// TwinCAT 3 PLC project PlcIotHttpSamplesTelegram
// ProgramVersion: 3.1.4026.25
// libraries:
//   Tc2_Standard, * (Beckhoff Automation GmbH)
//   Tc2_System, * (Beckhoff Automation GmbH)
//   Tc2_Utilities, * (Beckhoff Automation GmbH)
//   Tc3_IotBase, * (Beckhoff Automation GmbH)
//   Tc3_JsonXml, * (Beckhoff Automation GmbH)
//   Tc3_Module, * (Beckhoff Automation GmbH)
// project tree:
//   / PlcTask.TcTTO
//   POUs/ MAIN.TcPOU
//   POUs/Telegram/ FB_TestHTTP_Get_Telegram.TcPOU
// real-time tasks:
//   TASK PlcTask: cycle T#10ms, priority 25, ADS port 350

CONFIGURATION PlcIotHttpSamplesTelegram
    RESOURCE PLC ON TwinCAT3
        TASK PlcTask(INTERVAL := T#10ms, PRIORITY := 25);
        PROGRAM MAIN WITH PlcTask : MAIN;
    END_RESOURCE
END_CONFIGURATION

// ---- POUs/MAIN.TcPOU
PROGRAM MAIN
VAR
	// trigger command execution for Telegram samples
	bGetTelegram					: BOOL;

	fbHttpClientTelegram			: FB_IotHttpClient :=(sHostName := 'api.telegram.org',
									bKeepAlive := FALSE, tConnectionTimeout := T#10S);

	fbHttpGetTelegram				: FB_TestHTTP_Get_Telegram;
	sMessage						: STRING(500) := 'Hello from TwinCAT';
END_VAR

// init client parameters at startup
IF NOT fbHttpClientTelegram.bConfigured THEN
	fbHttpClientTelegram.nHostPort := 443;
	fbHttpClientTelegram.stTLS.bNoServerCertCheck := TRUE;
END_IF

IF fbHttpClientTelegram.bConfigured THEN
	fbHttpGetTelegram(bSend := bGetTelegram, fbClient := fbHttpClientTelegram, sMessage := sMessage);
END_IF

fbHttpClientTelegram.Execute();

END_PROGRAM

// ---- POUs/Telegram/FB_TestHTTP_Get_Telegram.TcPOU
FUNCTION_BLOCK FB_TestHTTP_Get_Telegram
VAR_INPUT
	bSend				: BOOL;
	sMessage			: STRING(500);
END_VAR
VAR_IN_OUT
	fbClient			: FB_IotHttpClient;
END_VAR
VAR_OUTPUT
	bBusy				: BOOL;
	bError				: BOOL;
END_VAR
VAR
	fbRequest			: FB_IotHttpRequest;
	fbJson				: FB_JsonDomParser;
	nState				: UDINT;
	RisingEdge			: R_TRIG;
	
	bGetContentResult	: BOOL;
	sContent			: STRING(511);
	
	bGetJsonResult		: BOOL;
	jsonDoc				: SJsonValue;
	
	nReqCount			: UDINT;	
	nResCount			: UDINT;
	nValidResCount		: UDINT;
	nErrCount			: UDINT;
	fbFormatString		: FB_FormatString;
	sBotApiKey			: STRING(500):='1644750049:AAH-censored_9RQkjlZ2IURbZWM';
	sChatId				: STRING(500):='114042censored';
	sConMessage			: STRING(500);
END_VAR

RisingEdge(CLK := bSend );

fbFormatString(
	sFormat	:= '/bot%s/sendMessage?chat_id=%s&text=%s', 
	arg1	:= F_STRING(sBotApiKey), 
	arg2	:= F_STRING(sChatId), 
	arg3	:= F_STRING(sMessage), 
	bError	=> , 
	nErrId	=> , 
	sOut	=> sConMessage);

CASE nState OF
0:	
	IF RisingEdge.Q THEN 
		IF fbRequest.SendRequest(sUri := sConMessage, fbClient := fbClient, eRequestType := ETcIotHttpRequestType.HTTP_GET, 0, 0, 0) THEN				
			nState := 1;
			nReqCount := nReqCount +1;
			bBusy := TRUE;
			bError := FALSE;
		END_IF					
	END_IF
1:
	IF NOT fbRequest.bBusy THEN
		bError := TRUE;
		IF NOT fbRequest.bError THEN				 
			// As an alternative to GetJsonDomContent, GetContent could be used				 
			// bGetContentResult := fbRequest.GetContent(pContent := ADR(sContent), nContentSize := SIZEOF(sContent), bSetNullTermination := TRUE);
			IF fbRequest.nStatusCode >= 200 AND fbRequest.nStatusCode < 300 THEN
				bGetJsonResult := FALSE;
				// Direct conversion into JSON object as the received message is in JSON format 
				jsonDoc := fbRequest.GetJsonDomContent(fbJson);
				IF jsonDoc <> 0 THEN
					; // do something with the response
					nValidResCount := nValidResCount+1;
					bError := FALSE;	
				END_IF							
				nResCount := nResCount +1;			
			END_IF
		END_IF
		nState := 0;
		bBusy := FALSE;
		IF bError THEN
			nErrCount := nErrCount +1;
		END_IF
	END_IF  	
END_CASE

END_FUNCTION_BLOCK
